{attribute 'qualified_only'}
{attribute 'strict'}
TYPE E_Message_OBC :
(
	eNoMessage := 0,
	eTooMuchOBC := 2,
	eExternalLockActive := 3,
	eErrorOBC := 4,
	eNoConnectionToBackend := 5
);
END_TYPE

(* stored: Version 1.1.0.1, ProductVersion 3.1.4024.6
   DUT E_Message_OBC: Id {9d416d8c-7fc1-47e9-8973-88aab371f411} *)
